(* IEC 61131-3 sources: AXOpen/src/components.keyence.vision/app/src/Documentation, 4 files *)

(* ---- Component_1.st ---- *)
USING AXOpen.Core;
NAMESPACE AXOpen.Components.Keyence.Vision
    {S7.extern=ReadWrite}
    CLASS Component_1 EXTENDS AXOpen.Core.AxoObject
        //<ComponentDeclaration>
        VAR PUBLIC
            Component : AXOpen.Components.Keyence.Vision.Axo_SR_750;
        END_VAR
        //</ComponentDeclaration>

        //<InitializationArgumentsDeclaration>
        VAR PUBLIC
            {#ix-set:AttributeName = "<#Activate manual control#>"}
            ActivateManualControl : BOOL;
        END_VAR
        //</InitializationArgumentsDeclaration>

        METHOD PUBLIC OVERRIDE Run
            VAR_INPUT
                inParent : IAxoObject;
            END_VAR

            SUPER.Run(inParent);

            IF ActivateManualControl THEN
                Component.ActivateManualControl();
            END_IF;

            //<Initialization>
            Component.Run(
                                parent                                          :=   THIS,
                                hwID                                            :=   HwIdentifiers#keyence_sr_750_HwID);
            //</Initialization>

            THIS.UseInSequencer();
        END_METHOD

        //<Usage>
        VAR PUBLIC
            Sequencer : AxoSequencer;
            Steps : ARRAY[0..3] OF AXOpen.Core.AxoStep;
        END_VAR

        VAR PRIVATE
            _ResultData  :   AXOpen.Components.Keyence.Vision.Axo_SR_750_ResultData;
        END_VAR

        METHOD PRIVATE UseInSequencer

            Sequencer.Run(THIS);
            Sequencer.Open();

            IF(Steps[0].Execute(Sequencer, 'Clear result data')) THEN
                IF(Component.ClearResultData().IsDone()) THEN
                    Sequencer.MoveNext();
                END_IF;
            END_IF;

            IF(Steps[1].Execute(Sequencer, 'Tune')) THEN
                IF(Component.Tune(UINT#0).IsDone()) THEN
                    Sequencer.MoveNext();
                END_IF;
            END_IF;

            IF(Steps[2].Execute(Sequencer, 'Read data')) THEN
                IF(Component.Read(UINT#0).IsDone()) THEN
                    Sequencer.MoveNext();
                END_IF;
            END_IF;

            IF(Steps[3].Execute(Sequencer, 'Evaluate data')) THEN
                _ResultData := Component.ResultData;
                Sequencer.CompleteSequence();
            END_IF;

        END_METHOD
        //</Usage>
    END_CLASS
END_NAMESPACE

(* ---- Component_2.st ---- *)
USING AXOpen.Core;
NAMESPACE AXOpen.Components.Keyence.Vision
    {S7.extern=ReadWrite}
    CLASS Component_2 EXTENDS AXOpen.Core.AxoObject
        //<ComponentDeclaration>
        VAR PUBLIC
            Component : AXOpen.Components.Keyence.Vision.Axo_SR_1000;
        END_VAR
        //</ComponentDeclaration>

        //<InitializationArgumentsDeclaration>
        VAR PUBLIC
            {#ix-set:AttributeName = "<#Activate manual control#>"}
            ActivateManualControl : BOOL;
        END_VAR
        //</InitializationArgumentsDeclaration>

        METHOD PUBLIC OVERRIDE Run
            VAR_INPUT
                inParent : IAxoObject;
            END_VAR

            SUPER.Run(inParent);

            IF ActivateManualControl THEN
                Component.ActivateManualControl();
            END_IF;

            //<Initialization>
            Component.Run(      parent                                          :=   THIS,
                                hwID                                            :=   HwIdentifiers#keyence_sr_1000_HwID);
            //</Initialization>

            THIS.UseInSequencer();
        END_METHOD

        //<Usage>
        VAR PUBLIC
            Sequencer : AxoSequencer;
            Steps : ARRAY[0..3] OF AXOpen.Core.AxoStep;
        END_VAR

        VAR PRIVATE
            _ResultData  :   AXOpen.Components.Keyence.Vision.Axo_SR_1000_ResultData;
        END_VAR

        METHOD PRIVATE UseInSequencer

            Sequencer.Run(THIS);
            Sequencer.Open();

            IF(Steps[0].Execute(Sequencer, 'Clear result data')) THEN
                IF(Component.ClearResultData().IsDone()) THEN
                    Sequencer.MoveNext();
                END_IF;
            END_IF;

            IF(Steps[1].Execute(Sequencer, 'Tune')) THEN
                IF(Component.Tune(UINT#0).IsDone()) THEN
                    Sequencer.MoveNext();
                END_IF;
            END_IF;

            IF(Steps[2].Execute(Sequencer, 'Read data')) THEN
                IF(Component.Read(UINT#0).IsDone()) THEN
                    Sequencer.MoveNext();
                END_IF;
            END_IF;

            IF(Steps[3].Execute(Sequencer, 'Evaluate data')) THEN
                _ResultData := Component.ResultData;
                Sequencer.CompleteSequence();
            END_IF;

        END_METHOD
        //</Usage>
    END_CLASS
END_NAMESPACE

(* ---- Component_3.st ---- *)
USING AXOpen.Core;
NAMESPACE AXOpen.Components.Keyence.Vision
    {S7.extern=ReadWrite}
    CLASS Component_3 EXTENDS AXOpen.Core.AxoObject
        //<ComponentDeclaration>
        VAR PUBLIC
            Component : AXOpen.Components.Keyence.Vision.Axo_IV3;
        END_VAR
        //</ComponentDeclaration>

        //<InitializationArgumentsDeclaration>
        VAR PUBLIC
            {#ix-set:AttributeName = "<#Activate manual control#>"}
            ActivateManualControl : BOOL;
        END_VAR
        //</InitializationArgumentsDeclaration>

        METHOD PUBLIC OVERRIDE Run
            VAR_INPUT
                inParent : IAxoObject;
            END_VAR

            SUPER.Run(inParent);

            IF ActivateManualControl THEN
                Component.ActivateManualControl();
            END_IF;

            //<Initialization>
            Component.Run(      parent                                          :=   THIS,
                                hwID                                            :=   HwIdentifiers#keyence_iv3_HwID);
            //</Initialization>

            THIS.UseInSequencer();
        END_METHOD

        //<Usage>
        VAR PUBLIC
            Sequencer : AxoSequencer;
            Steps : ARRAY[0..3] OF AXOpen.Core.AxoStep;
        END_VAR

        VAR PRIVATE
            _OverAllResult  : BOOL;
            _ResultData  :  ARRAY[0..20] OF UINT;
        END_VAR

        METHOD PRIVATE UseInSequencer

            Sequencer.Run(THIS);
            Sequencer.Open();

            IF(Steps[0].Execute(Sequencer, 'Restore')) THEN
                Component.Restore();
                Sequencer.MoveNext();
            END_IF;

            IF(Steps[1].Execute(Sequencer, 'Change program')) THEN
                IF(Component.ChangeProgram(UINT#0).IsDone()) THEN
                    Sequencer.MoveNext();
                END_IF;
            END_IF;

            IF(Steps[2].Execute(Sequencer, 'Trigger')) THEN
                IF(Component.Trigger().IsDone()) THEN
                    Sequencer.MoveNext();
                END_IF;
            END_IF;

            IF(Steps[3].Execute(Sequencer, 'Access the result data')) THEN
                _OverAllResult := Component.Inputs.DeviceResultBits_1.OverallJudgmentOK;
                // The meaning of the result data changes with the type of the control,
                // so it must be evaluated individually in the production code
                _ResultData[0] := Component.Inputs.ToolResult_1.MatchingRate;
                _ResultData[1] := Component.Inputs.ToolResult_1.MatchingRateMAX;
                _ResultData[2] := Component.Inputs.ToolResult_1.MatchingRateMIN;
                _ResultData[3] := Component.Inputs.ToolResult_1.LowerThreshold;
                _ResultData[4] := Component.Inputs.ToolResult_1.UpperThreshold;
                _ResultData[5] := Component.Inputs.ToolResult_1.DecimalPointPosition;
                _ResultData[6] := Component.Inputs.ToolResult_1.Data_1;
                _ResultData[7] := Component.Inputs.ToolResult_1.Data_2;
                _ResultData[8] := Component.Inputs.ToolResult_1.Data_3;
                Sequencer.CompleteSequence();
            END_IF;

        END_METHOD
        //</Usage>
    END_CLASS
END_NAMESPACE

(* ---- DocumentationContext.st ---- *)
NAMESPACE AXOpen.Components.Keyence.Vision
    {S7.extern=ReadWrite}
    CLASS DocumentationContext EXTENDS AXOpen.Core.AxoContext
        VAR PUBLIC
            rootObject      : AxoObject;
            componentOne    : AXOpen.Components.Keyence.Vision.Component_1;
            componentTwo    : AXOpen.Components.Keyence.Vision.Component_2;
            componentThree  : AXOpen.Components.Keyence.Vision.Component_3;
        END_VAR

        METHOD PROTECTED OVERRIDE Main
            THIS.InitializeRootObject(rootObject);
            componentOne.Run(rootObject);
            componentTwo.Run(rootObject);
            componentThree.Run(rootObject);
        END_METHOD
    END_CLASS
END_NAMESPACE
